% RSLogix 500 project DDE MESSAGING_BAK004.RSS, saved by version 8.30.00.16 %
PROJECT "UNTITLED"    % processor: Bul.1763 MicroLogix 1100 Series B %

PROGRAM FILES
  LAD 2   11 rungs

DATA FILES
  O0 OUTPUT  4 elements
  I1 INPUT  6 elements
  S2 STATUS  66 elements
  B3 BINARY  2 elements
  T4 TIMER  1 elements
  C5 COUNTER  1 elements
  R6 CONTROL  1 elements
  N7 INTEGER  5 elements
  F8 FLOAT  1 elements
  ST9 STRING  8 elements

LADDER 2
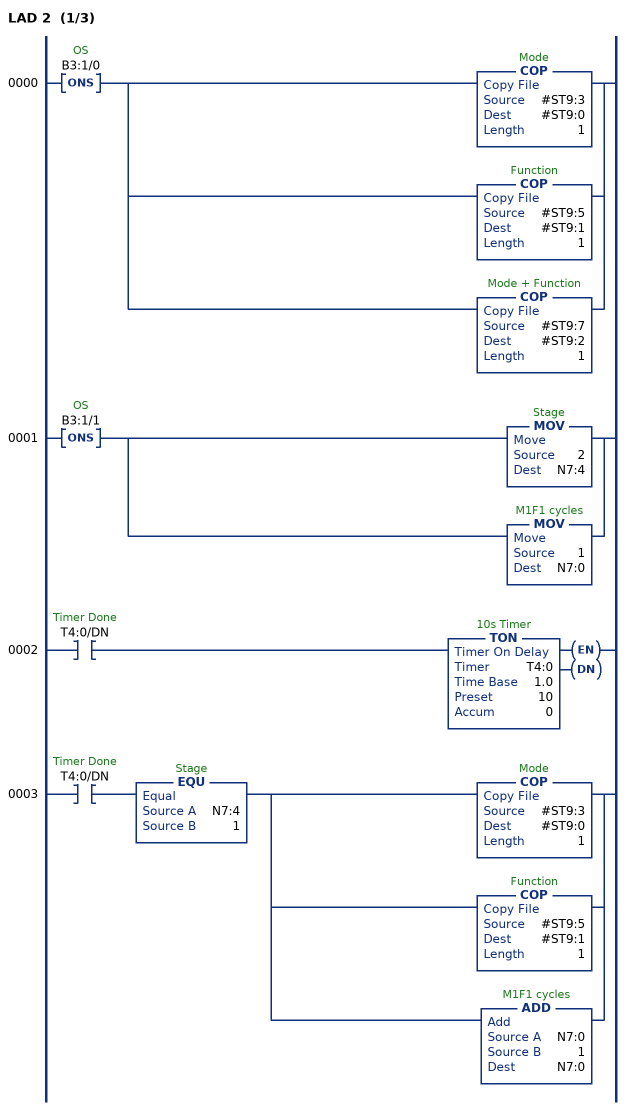
% Rung: 0 %
SOR ONS B3:1/0 BST COP #ST9:3 #ST9:0 1 NXB BST COP #ST9:5 #ST9:1 1 NXB COP #ST9:7 #ST9:2 1 BND BND EOR
%   B3:1/0  "OS" %
%   ST9:3  "Mode-1" %
%   ST9:0  "Mode" %
%   ST9:5  "F1" %
%   ST9:1  "Function" %
%   ST9:7  "Mode-1,F1" %
%   ST9:2  "Mode + Function" %
% Rung: 1 %
SOR ONS B3:1/1 BST MOV 2 N7:4 NXB MOV 1 N7:0 BND EOR
%   B3:1/1  "OS" %
%   N7:4  "Stage" %
%   N7:0  "M1F1 cycles" %
% Rung: 2 %
SOR XIC T4:0/DN TON T4:0 1.0 10 0 EOR
%   T4:0/DN  "Timer Done" %
%   T4:0  "10s Timer" %
% Rung: 3 %
SOR XIC T4:0/DN EQU N7:4 1 BST COP #ST9:3 #ST9:0 1 NXB BST COP #ST9:5 #ST9:1 1 NXB ADD N7:0 1 N7:0 BND BND EOR
%   T4:0/DN  "Timer Done" %
%   N7:4  "Stage" %
%   ST9:3  "Mode-1" %
%   ST9:0  "Mode" %
%   ST9:5  "F1" %
%   ST9:1  "Function" %
%   N7:0  "M1F1 cycles" %

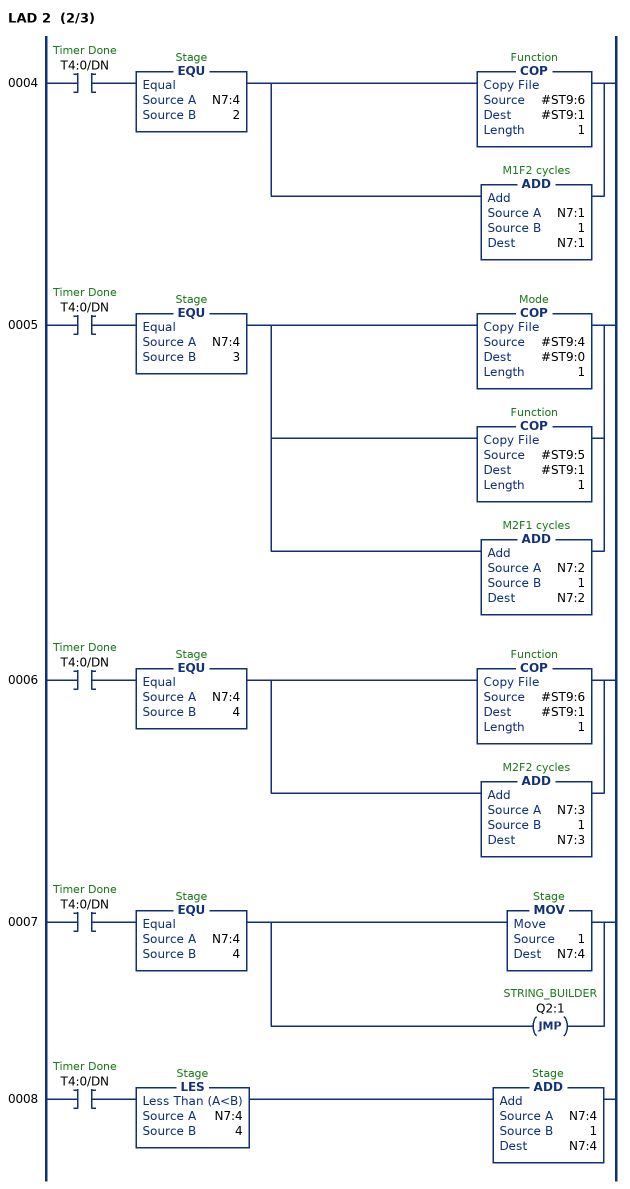
% Rung: 4 %
SOR XIC T4:0/DN EQU N7:4 2 BST COP #ST9:6 #ST9:1 1 NXB ADD N7:1 1 N7:1 BND EOR
%   T4:0/DN  "Timer Done" %
%   N7:4  "Stage" %
%   ST9:6  "F2" %
%   ST9:1  "Function" %
%   N7:1  "M1F2 cycles" %
% Rung: 5 %
SOR XIC T4:0/DN EQU N7:4 3 BST COP #ST9:4 #ST9:0 1 NXB BST COP #ST9:5 #ST9:1 1 NXB ADD N7:2 1 N7:2 BND BND EOR
%   T4:0/DN  "Timer Done" %
%   N7:4  "Stage" %
%   ST9:4  "Mode-2" %
%   ST9:0  "Mode" %
%   ST9:5  "F1" %
%   ST9:1  "Function" %
%   N7:2  "M2F1 cycles" %
% Rung: 6 %
SOR XIC T4:0/DN EQU N7:4 4 BST COP #ST9:6 #ST9:1 1 NXB ADD N7:3 1 N7:3 BND EOR
%   T4:0/DN  "Timer Done" %
%   N7:4  "Stage" %
%   ST9:6  "F2" %
%   ST9:1  "Function" %
%   N7:3  "M2F2 cycles" %
% Rung: 7 %
SOR XIC T4:0/DN EQU N7:4 4 BST MOV 1 N7:4 NXB JMP Q2:1 BND EOR
%   T4:0/DN  "Timer Done" %
%   N7:4  "Stage" %
%   Q2:1  STRING_BUILDER %
% Rung: 8 %
SOR XIC T4:0/DN LES N7:4 4 ADD N7:4 1 N7:4 EOR
%   T4:0/DN  "Timer Done" %
%   N7:4  "Stage" %

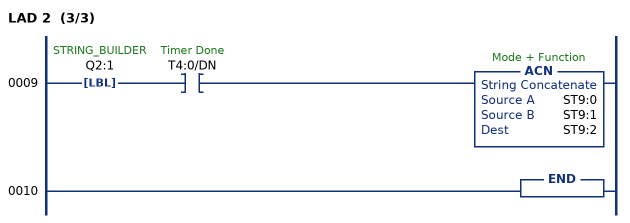
% Rung: 9 %
SOR LBL Q2:1 XIC T4:0/DN ACN ST9:0 ST9:1 ST9:2 EOR
%   Q2:1  STRING_BUILDER %
%   T4:0/DN  "Timer Done" %
%   ST9:0  "Mode" %
%   ST9:1  "Function" %
%   ST9:2  "Mode + Function" %
% Rung: 10 %
SOR END EOR

OTHER DOCUMENTED ADDRESSES
  B3:0/0  "Trigger"
  B3:0/1  "Reset"
  ST9:8  "Mode-1,F1"

DATA TABLE (non-zero values as saved)
DATA T4
% .PRE .ACC %
% T4:0 % 10 0
